{attribute 'GeneratedUsingTerminal: EP2339-0042-0018'}
{attribute addProperty BoxType "EP2339-0042-0018"}
{attribute addProperty Description "EP2339-0042 16 Ch. Dig. Input/Output 24V, 0.5A, M12 "}
{attribute addProperty Physics "YY"}
{attribute addProperty Id "DI_X01_4AT %I*DI_X_830843C11DI_X01_2AT %I*DI_X_830843C11DI_X02_4AT %I*DI_X_830843C11DI_X02_2AT %I*DI_X_830843C11DI_X03_4AT %I*DI_X_830843C11DI_X03_2AT %I*DI_X_830843C11DI_X04_4AT %I*DI_X_830843C11DI_X04_2AT %I*DI_X_830843C11DI_X05_4AT %I*DI_X_830843C11DI_X05_2AT %I*DI_X_830843C11DI_X06_4AT %I*DI_X_830843C11DI_X06_2AT %I*DI_X_830843C11DI_X07_4AT %I*DI_X_830843C11DI_X07_2AT %I*DI_X_830843C11DI_X08_4AT %I*DI_X_830843C11DI_X08_2AT %I*DI_X_830843C11DO_X01_4AT %Q*DO_X_42CA91F71DO_X01_2AT %Q*DO_X_42CA91F71DO_X02_4AT %Q*DO_X_42CA91F71DO_X02_2AT %Q*DO_X_42CA91F71DO_X03_4AT %Q*DO_X_42CA91F71DO_X03_2AT %Q*DO_X_42CA91F71DO_X04_4AT %Q*DO_X_42CA91F71DO_X04_2AT %Q*DO_X_42CA91F71DO_X05_4AT %Q*DO_X_42CA91F71DO_X05_2AT %Q*DO_X_42CA91F71DO_X06_4AT %Q*DO_X_42CA91F71DO_X06_2AT %Q*DO_X_42CA91F71DO_X07_4AT %Q*DO_X_42CA91F71DO_X07_2AT %Q*DO_X_42CA91F71DO_X08_4AT %Q*DO_X_42CA91F71DO_X08_2AT %Q*DO_X_42CA91F71WcStateAT %I*WcState_9091E0EB2InfoDataAT %I*InfoData_6F19DB2B2"}
{attribute addProperty CRC "3818076209"}
{attribute addProperty Size "36"}
TYPE EP2339_E3933831 EXTENDS EtcSlaveBoxBase_77A0E4A7 :
STRUCT
	{attribute addProperty Name "DI_X01_4"}
	DI_X01_4 : DI_X_830843C1;
	{attribute addProperty Name "DI_X01_2"}
	DI_X01_2 : DI_X_830843C1;
	{attribute addProperty Name "DI_X02_4"}
	DI_X02_4 : DI_X_830843C1;
	{attribute addProperty Name "DI_X02_2"}
	DI_X02_2 : DI_X_830843C1;
	{attribute addProperty Name "DI_X03_4"}
	DI_X03_4 : DI_X_830843C1;
	{attribute addProperty Name "DI_X03_2"}
	DI_X03_2 : DI_X_830843C1;
	{attribute addProperty Name "DI_X04_4"}
	DI_X04_4 : DI_X_830843C1;
	{attribute addProperty Name "DI_X04_2"}
	DI_X04_2 : DI_X_830843C1;
	{attribute addProperty Name "DI_X05_4"}
	DI_X05_4 : DI_X_830843C1;
	{attribute addProperty Name "DI_X05_2"}
	DI_X05_2 : DI_X_830843C1;
	{attribute addProperty Name "DI_X06_4"}
	DI_X06_4 : DI_X_830843C1;
	{attribute addProperty Name "DI_X06_2"}
	DI_X06_2 : DI_X_830843C1;
	{attribute addProperty Name "DI_X07_4"}
	DI_X07_4 : DI_X_830843C1;
	{attribute addProperty Name "DI_X07_2"}
	DI_X07_2 : DI_X_830843C1;
	{attribute addProperty Name "DI_X08_4"}
	DI_X08_4 : DI_X_830843C1;
	{attribute addProperty Name "DI_X08_2"}
	DI_X08_2 : DI_X_830843C1;
	{attribute addProperty Name "DO_X01_4"}
	DO_X01_4 : DO_X_42CA91F7;
	{attribute addProperty Name "DO_X01_2"}
	DO_X01_2 : DO_X_42CA91F7;
	{attribute addProperty Name "DO_X02_4"}
	DO_X02_4 : DO_X_42CA91F7;
	{attribute addProperty Name "DO_X02_2"}
	DO_X02_2 : DO_X_42CA91F7;
	{attribute addProperty Name "DO_X03_4"}
	DO_X03_4 : DO_X_42CA91F7;
	{attribute addProperty Name "DO_X03_2"}
	DO_X03_2 : DO_X_42CA91F7;
	{attribute addProperty Name "DO_X04_4"}
	DO_X04_4 : DO_X_42CA91F7;
	{attribute addProperty Name "DO_X04_2"}
	DO_X04_2 : DO_X_42CA91F7;
	{attribute addProperty Name "DO_X05_4"}
	DO_X05_4 : DO_X_42CA91F7;
	{attribute addProperty Name "DO_X05_2"}
	DO_X05_2 : DO_X_42CA91F7;
	{attribute addProperty Name "DO_X06_4"}
	DO_X06_4 : DO_X_42CA91F7;
	{attribute addProperty Name "DO_X06_2"}
	DO_X06_2 : DO_X_42CA91F7;
	{attribute addProperty Name "DO_X07_4"}
	DO_X07_4 : DO_X_42CA91F7;
	{attribute addProperty Name "DO_X07_2"}
	DO_X07_2 : DO_X_42CA91F7;
	{attribute addProperty Name "DO_X08_4"}
	DO_X08_4 : DO_X_42CA91F7;
	{attribute addProperty Name "DO_X08_2"}
	DO_X08_2 : DO_X_42CA91F7;
	{attribute addProperty Name "WcState"}
	WcState : WcState_9091E0EB;
	{attribute addProperty Name "InfoData"}
	InfoData : InfoData_6F19DB2B;
END_STRUCT
END_TYPE

(* stored: Version 1.2.0.0, ProductVersion 3.1.4024.9
   DUT EP2339_E3933831: Id {886894cf-f2d6-49c1-9d8f-eafeaad4c084} *)
